FUNCTION SortMaterialPositionArray : BOOL
VAR_IN_OUT
	arr : ARRAY[*] OF MaterialPosition;
END_VAR
VAR
	//iterators
	i : INT;
	j : INT;
END_VAR

FOR i:=0 TO GVL.maxMaterials BY 1 DO
	FOR j:=0 TO GVL.maxMaterials BY 1 DO
		IF arr[j].position > arr[j+1].position THEN
			SwapMaterialPosition(ADR(arr[j]), ADR(arr[j+1]));
		END_IF
	END_FOR
END_FOR

END_FUNCTION

(* stored: Version 1.1.0.1, ProductVersion 3.1.4024.11
   POU SortMaterialPositionArray: Id {73245192-df11-4d1b-bad1-b2d9b4c81944}, SpecialFunc None *)
